// TIA Portal V16 export
// export: Created 2021-09-08T12:46:12.106135Z, ExportSetting WithDefaults, DisplayName Totally Integrated Automation Portal, DisplayVersion V16 Update 3, DisplayName TIA Portal Version Control Interface, DisplayVersion V16 Update 2, DisplayName TIA Portal Openness, DisplayVersion V16 Update 3, DisplayName TIA Portal Teamcenter Gateway, DisplayVersion V16, DisplayName STEP 7 Professional, DisplayVersion V16 Update 3, DisplayName STEP 7 Safety, DisplayVersion V16, DisplayName WinCC Advanced, DisplayVersion V16 Update 3
DATA_BLOCK "dtPID"   // DB8
{ S7_Optimized_Access := 'FALSE' }
VERSION : 0.1
// stored: AutoNumber true, DBAccessibleFromOPCUA true, IsOnlyStoredInLoadMemory false, IsWriteProtectedInAS false
   VAR RETAIN
      pidP30x : "setPID";
      pidP120x { S7_SetPoint := 'True'} : "setPID";
      pidP150x { S7_SetPoint := 'True'} : "setPID";
      pidP901 { S7_SetPoint := 'True'} : "setPID";
      pidP1301 { S7_SetPoint := 'True'} : "setPID";
   END_VAR
BEGIN
END_DATA_BLOCK
